# EPICS autosave request: iocs/peakAnalyserIOC/iocBoot/iocPeakAnalyser/auto_settings.req
file "peakAnalyser_settings.req",   P=$(P),  R=cam1:
file "NDStdArrays_settings.req",    P=$(P),  R=image1:
file "commonPlugin_settings.req",   P=$(P)
